Universal Robots PolyScope program: 111.urp

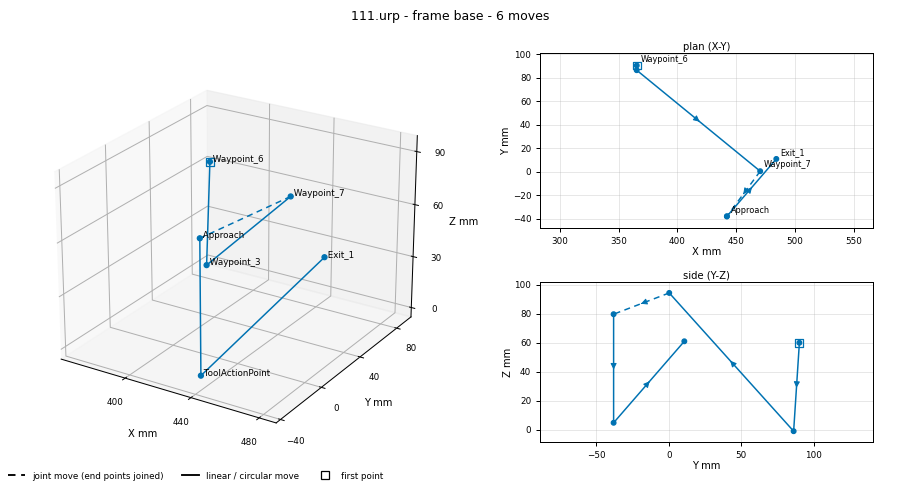
[picture p0: tool path of 111.urp in frame base, 6 of 6 moves have a stored position in this frame; points joined in program order, loops and branches not executed]
Program 111 (installation=default directory=/programs createdIn=5.11.9.1010452 lastSavedIn=5.11.9.1010452 robotSerialNumber=20225200364)
Calibrated DH parameters: a=[0.000056, -0.511675, -0.549032, 0.000082, -0.00003, 0]; d=[0.180587, -182.578947, 231.390066, -48.637383, 0.119742, 0.115539]; alpha=[1.571438, -0.00184, 0.003237, 1.569836, -1.571354, 0]; deltaTheta=[-0.000001, 0.580933, 5.982442, -0.280193, -0.000002, 0]
Robot Program (runOnlyOnce=false)
  URCap RG Grip (OnRobot, OnRobot A/S) dataModel(rg-target-force=40.0, rg-target-width=0.0386)
  MoveL speed 250 mm/s, acceleration 1200 mm/s^2 (useActiveTCP=true) feature=Base
    Waypoint Waypoint_6: TCP in base x=365.397 y=90.243 z=59.995 mm, rx=2.2777 ry=-2.1609 rz=0.0005 rad; joints [41.388, -66.204, -149.958, -53.913, 90.199, 38.438] deg; TCP offset x=0 y=0 z=228.6 mm, rx=0 ry=0 rz=0 rad
    Waypoint Waypoint_3: TCP in base x=365.344 y=86.267 z=-1.114 mm, rx=2.2779 ry=-2.1606 rz=0.0003 rad; joints [40.862, -74.238, -154.151, -41.693, 90.179, 37.946] deg
    Loop Forever
      Placeholder
    CallSubProgram
    URCap RG Grip (OnRobot, OnRobot A/S) dataModel(rg-target-force=40.0, rg-target-width=0.015700000000000002, Variable(key=on_return, variable(name=on_return)))
    Waypoint Waypoint_7: TCP in base x=470.463 y=0.3 z=94.424 mm, rx=2.2779 ry=-2.1606 rz=0.0002 rad; joints [21.723, -76.465, -139.77, -53.836, 90.159, 18.776] deg
  URCap Palletizing (polyscope-pallet-impl, Universal Robots) dataModel(palletFeature=Base, isPalletizing=true, Length(key=objectHeight value=0.012 unit=M), Variable(key=name, variable(name=Pallet_1)), Variable(key=globalCountingVariable, variable(name=Pallet_1_cnt, initializeExpression=1)), Variable(key=layerNumberVariable, variable(name=Pallet_1_lno, initializeExpression=1)), Variable(key=layerCountingVariable, variable(name=Pallet_1_lct, initializeExpression=1)), Variable(key=handleSeparatorVariable, variable(name=Pallet_1_sep, initializeExpression=False)), Variable(key=totalCountVariable, variable(name=Pallet_1_tct, initializeExpression=1)), Variable(key=referencePoint, variable(featureName=referencePoint)), Variable(key=separatorPoint, variable(featureName=separatorPoint))); state(isChildrenLocked=true)
    URCap Patterns (polyscope-pallet-impl, Universal Robots) state(isChildrenLocked=true)
      URCap Pattern (polyscope-pallet-impl, Universal Robots) dataModel(UUID=9b3320d7-96d8-4d83-b7ca-67031437823e, patternType=GRID, columns=3, rows=3, Variable(key=nameVariable, variable(name=Grid_Pattern_1))); state(isChildrenLocked=true)
        URCap Item (polyscope-pallet-impl, Universal Robots) dataModel(UUID=3edb64ea-5930-4200-949f-ba596bc77f3b, patternType=GRID, index=0, calibrationDeltaTheta=[-7.716858584048969E-7, 0.5809325624761351, 5.982441805008871, -0.2801932900558549, -2.087699179323388E-6, 7.182941588051994E-8], calibrationA=[5.584882619731399E-5, -0.5116748572506173, -0.549032347835167, 8.201669770320986E-5, -3.0447895639691726E-5, 0.0], calibrationD=[0.18058730552743416, -182.578946596082, 231.39006605348337, -48.6373829503458, 0.11974176219014578, 0.11553881708205978], calibrationAlpha=[1.5714381462339815, -0.001839843720035074, 0.003236774450590588, 1.5698364982897774, -1.571354041521518, 0.0], calibrationJointChecksum=[-1488423315, -1488334884, 658253144, -1490959501, -1490992896, -1492776484], calibrationStatus=2, calibrationValidChecksum=true, baseToFeature=[0.0, 0.0, 0.0, 0.0, 0.0, 0.0], TCPOffset=[1.394757124627971E-5, 5.864256917231803E-6, 0.2286062449034809, -1.5736321545787795E-5, 5.11290631336734E-5, -4.190407476781124E-5], Variable(key=variable, variable(name=CornerItem_1)), JointPositions(key=jointpositions, JointPosition(key=[1], Angle(key=pos value=0.315696 unit=RAD)), JointPosition(key=[2], Angle(key=pos value=-1.445177 unit=RAD)), JointPosition(key=[3], Angle(key=pos value=-2.574702 unit=RAD)), JointPosition(key=[4], Angle(key=pos value=-0.691948 unit=RAD)), JointPosition(key=[5], Angle(key=pos value=1.574025 unit=RAD)), JointPosition(key=[6], Angle(key=pos value=0.265625 unit=RAD))))
        URCap Item (polyscope-pallet-impl, Universal Robots) dataModel(UUID=12f326a5-259c-497f-afe2-b32ea041848a, patternType=GRID, index=1, calibrationDeltaTheta=[-7.716858584048969E-7, 0.5809325624761351, 5.982441805008871, -0.2801932900558549, -2.087699179323388E-6, 7.182941588051994E-8], calibrationA=[5.584882619731399E-5, -0.5116748572506173, -0.549032347835167, 8.201669770320986E-5, -3.0447895639691726E-5, 0.0], calibrationD=[0.18058730552743416, -182.578946596082, 231.39006605348337, -48.6373829503458, 0.11974176219014578, 0.11553881708205978], calibrationAlpha=[1.5714381462339815, -0.001839843720035074, 0.003236774450590588, 1.5698364982897774, -1.571354041521518, 0.0], calibrationJointChecksum=[-1488423315, -1488334884, 658253144, -1490959501, -1490992896, -1492776484], calibrationStatus=2, calibrationValidChecksum=true, baseToFeature=[0.0, 0.0, 0.0, 0.0, 0.0, 0.0], TCPOffset=[2.6395109693044816E-5, 5.65734824152786E-5, 0.2286631752094506, -1.3505097444767376E-4, 7.09143507036969E-5, 8.366689758555559E-6], Variable(key=variable, variable(name=CornerItem_2)), JointPositions(key=jointpositions, JointPosition(key=[1], Angle(key=pos value=0.254966 unit=RAD)), JointPosition(key=[2], Angle(key=pos value=-1.625257 unit=RAD)), JointPosition(key=[3], Angle(key=pos value=-2.405287 unit=RAD)), JointPosition(key=[4], Angle(key=pos value=-0.681283 unit=RAD)), JointPosition(key=[5], Angle(key=pos value=1.573736 unit=RAD)), JointPosition(key=[6], Angle(key=pos value=0.205114 unit=RAD))))
        URCap Item (polyscope-pallet-impl, Universal Robots) dataModel(UUID=9547d85f-1113-4171-9186-e072b20d7910, patternType=GRID, index=2, calibrationDeltaTheta=[-7.716858584048969E-7, 0.5809325624761351, 5.982441805008871, -0.2801932900558549, -2.087699179323388E-6, 7.182941588051994E-8], calibrationA=[5.584882619731399E-5, -0.5116748572506173, -0.549032347835167, 8.201669770320986E-5, -3.0447895639691726E-5, 0.0], calibrationD=[0.18058730552743416, -182.578946596082, 231.39006605348337, -48.6373829503458, 0.11974176219014578, 0.11553881708205978], calibrationAlpha=[1.5714381462339815, -0.001839843720035074, 0.003236774450590588, 1.5698364982897774, -1.571354041521518, 0.0], calibrationJointChecksum=[-1488423315, -1488334884, 658253144, -1490959501, -1490992896, -1492776484], calibrationStatus=2, calibrationValidChecksum=true, baseToFeature=[0.0, 0.0, 0.0, 0.0, 0.0, 0.0], TCPOffset=[7.665779734530864E-7, 2.0563258760764036E-5, 0.22859534913470098, 2.1874033595180868E-5, -3.4141777985640826E-7, -1.7572412885038355E-6], Variable(key=variable, variable(name=CornerItem_3)), JointPositions(key=jointpositions, JointPosition(key=[1], Angle(key=pos value=0.442273 unit=RAD)), JointPosition(key=[2], Angle(key=pos value=-1.623432 unit=RAD)), JointPosition(key=[3], Angle(key=pos value=-2.407279 unit=RAD)), JointPosition(key=[4], Angle(key=pos value=-0.681116 unit=RAD)), JointPosition(key=[5], Angle(key=pos value=1.573738 unit=RAD)), JointPosition(key=[6], Angle(key=pos value=0.39242 unit=RAD))))
        URCap Item (polyscope-pallet-impl, Universal Robots) dataModel(UUID=550561b9-d83e-4091-9ba4-89db74e54993, patternType=GRID, index=3, calibrationDeltaTheta=[-7.716858584048969E-7, 0.5809325624761351, 5.982441805008871, -0.2801932900558549, -2.087699179323388E-6, 7.182941588051994E-8], calibrationA=[5.584882619731399E-5, -0.5116748572506173, -0.549032347835167, 8.201669770320986E-5, -3.0447895639691726E-5, 0.0], calibrationD=[0.18058730552743416, -182.578946596082, 231.39006605348337, -48.6373829503458, 0.11974176219014578, 0.11553881708205978], calibrationAlpha=[1.5714381462339815, -0.001839843720035074, 0.003236774450590588, 1.5698364982897774, -1.571354041521518, 0.0], calibrationJointChecksum=[-1488423315, -1488334884, 658253144, -1490959501, -1490992896, -1492776484], calibrationStatus=2, calibrationValidChecksum=true, baseToFeature=[0.0, 0.0, 0.0, 0.0, 0.0, 0.0], TCPOffset=[3.3147242760801776E-5, 4.284661143133528E-5, 0.22863601896981714, -6.334259502335585E-5, 3.6431845443588446E-5, 3.4181487431328425E-6], Variable(key=variable, variable(name=CornerItem_4)), JointPositions(key=jointpositions, JointPosition(key=[1], Angle(key=pos value=0.539602 unit=RAD)), JointPosition(key=[2], Angle(key=pos value=-1.445948 unit=RAD)), JointPosition(key=[3], Angle(key=pos value=-2.574215 unit=RAD)), JointPosition(key=[4], Angle(key=pos value=-0.691816 unit=RAD)), JointPosition(key=[5], Angle(key=pos value=1.574025 unit=RAD)), JointPosition(key=[6], Angle(key=pos value=0.48954 unit=RAD))))
    URCap Layers (polyscope-pallet-impl, Universal Robots) dataModel(separators=[false], selectedPatterns=[9b3320d7-96d8-4d83-b7ca-67031437823e])
    URCap At Each Item (polyscope-pallet-impl, Universal Robots) dataModel(selectedPattern=9b3320d7-96d8-4d83-b7ca-67031437823e, selectedPosition=3edb64ea-5930-4200-949f-ba596bc77f3b, Approach_calibrationDeltaTheta=[-7.716858584048969E-7, 0.5809325624761351, 5.982441805008871, -0.2801932900558549, -2.087699179323388E-6, 7.182941588051994E-8], Approach_calibrationA=[5.584882619731399E-5, -0.5116748572506173, -0.549032347835167, 8.201669770320986E-5, -3.0447895639691726E-5, 0.0], Approach_calibrationD=[0.18058730552743416, -182.578946596082, 231.39006605348337, -48.6373829503458, 0.11974176219014578, 0.11553881708205978], Approach_calibrationAlpha=[1.5714381462339815, -0.001839843720035074, 0.003236774450590588, 1.5698364982897774, -1.571354041521518, 0.0], Approach_calibrationJointChecksum=[-1488423315, -1488334884, 658253144, -1490959501, -1490992896, -1492776484], Approach_calibrationStatus=2, Approach_calibrationValidChecksum=true, Approach_baseToFeature=[0.0, 0.0, 0.0, 0.0, 0.0, 0.0], Approach_TCPOffset=[-9.57256240663451E-8, -1.147904522547094E-6, 0.22860158750770332, 1.2097467679843313E-5, 2.4606278618820782E-5, -6.197340490944416E-5], Exit_calibrationDeltaTheta=[-7.716858584048969E-7, 0.5809325624761351, 5.982441805008871, -0.2801932900558549, -2.087699179323388E-6, 7.182941588051994E-8], Exit_calibrationA=[5.584882619731399E-5, -0.5116748572506173, -0.549032347835167, 8.201669770320986E-5, -3.0447895639691726E-5, 0.0], Exit_calibrationD=[0.18058730552743416, -182.578946596082, 231.39006605348337, -48.6373829503458, 0.11974176219014578, 0.11553881708205978], Exit_calibrationAlpha=[1.5714381462339815, -0.001839843720035074, 0.003236774450590588, 1.5698364982897774, -1.571354041521518, 0.0], Exit_calibrationJointChecksum=[-1488423315, -1488334884, 658253144, -1490959501, -1490992896, -1492776484], Exit_calibrationStatus=2, Exit_calibrationValidChecksum=true, Exit_baseToFeature=[0.0, 0.0, 0.0, 0.0, 0.0, 0.0], Exit_TCPOffset=[3.093053591055571E-5, 3.5837716356124094E-5, 0.2286459449007466, -8.649023224774153E-5, 6.489381906908273E-5, -1.5644032707469721E-6], currentWizardState=LANDING, Pose(key=refBaseToFeature, Position(key=posePosition, Length(key=X value=0 unit=M), Length(key=Y value=0 unit=M), Length(key=Z value=0 unit=M)), Rotation(key=poseRotation, Angle(key=RX value=0 unit=RAD), Angle(key=RY value=0 unit=RAD), Angle(key=RZ value=0 unit=RAD))), Pose(key=refPose, Position(key=posePosition, Length(key=X value=0.442114 unit=M), Length(key=Y value=-0.038132 unit=M), Length(key=Z value=0.004708 unit=M)), Rotation(key=poseRotation, Angle(key=RX value=2.278814 unit=RAD), Angle(key=RY value=-2.162479 unit=RAD), Angle(key=RZ value=0.000041 unit=RAD))), JointPositions(key=Approach_jointpositions, JointPosition(key=[1], Angle(key=pos value=0.31587 unit=RAD)), JointPosition(key=[2], Angle(key=pos value=-1.296314 unit=RAD)), JointPosition(key=[3], Angle(key=pos value=-2.497338 unit=RAD)), JointPosition(key=[4], Angle(key=pos value=-0.918205 unit=RAD)), JointPosition(key=[5], Angle(key=pos value=1.574515 unit=RAD)), JointPosition(key=[6], Angle(key=pos value=0.264918 unit=RAD))), JointPositions(key=Exit_jointpositions, JointPosition(key=[1], Angle(key=pos value=0.388557 unit=RAD)), JointPosition(key=[2], Angle(key=pos value=-1.416971 unit=RAD)), JointPosition(key=[3], Angle(key=pos value=-2.454659 unit=RAD)), JointPosition(key=[4], Angle(key=pos value=-0.840229 unit=RAD)), JointPosition(key=[5], Angle(key=pos value=1.574261 unit=RAD)), JointPosition(key=[6], Angle(key=pos value=0.337995 unit=RAD))))
      URCap Generated Movements (polyscope-pallet-impl, Universal Robots) state(isChildrenLocked=true)
        MoveJ speed 60 deg/s, acceleration 80 deg/s^2 (useActiveTCP=true) feature=referencePoint
          Waypoint Approach: TCP in base x=442.115 y=-38.132 z=79.734 mm, rx=2.2789 ry=-2.1624 rz=0.0001 rad; joints [18.06, -109.002, -152.076, -8.891, 90.063, 15.271] deg; TCP offset x=0 y=0 z=0 mm, rx=0 ry=0 rz=0 rad; feature pose in base x=442.114 y=-38.132 z=4.708 mm, rx=2.2788 ry=-2.1625 rz=0 rad
        MoveL speed 250 mm/s, acceleration 1200 mm/s^2 (useActiveTCP=true) feature(featureName=referencePoint)
          Waypoint ToolActionPoint: TCP in base x=442.114 y=-38.132 z=4.708 mm, rx=2.2788 ry=-2.1625 rz=0 rad; joints [18.047, -123.844, -151.479, 5.354, 89.994, 15.278] deg; TCP offset x=0 y=0 z=0 mm, rx=0 ry=0 rz=0 rad
        Folder Tool action
          URCap RG Grip (OnRobot, OnRobot A/S) dataModel(rg-target-force=40.0, rg-target-width=0.0386)
        MoveL speed 250 mm/s, acceleration 1200 mm/s^2 (useActiveTCP=true) feature(featureName=referencePoint)
          Waypoint Exit_1: TCP in base x=484.179 y=10.734 z=61.01 mm, rx=2.2787 ry=-2.1624 rz=0 rad; joints [22.227, -113.692, -147.68, -8.603, 90.054, 19.444] deg; TCP offset x=0 y=0 z=0 mm, rx=0 ry=0 rz=0 rad
